FUNCTION AddToBundlesArray : BOOL
VAR_INPUT
	arr : POINTER TO Bundle;
	
END_VAR
VAR
END_VAR

FOR i:=0 TO CONSTS.maxQueue BY 1 DO
	IF BundleIsValid(bundlesQueue[i]) AND NOT bundlesBypass[i] THEN
		bundlesQueue[i] := bundleIn;
		bundlesBypass[i] := FALSE;
		
		receive := TRUE;
		RETURN;
	END_IF
END_FOR

END_FUNCTION

(* stored: Version 1.1.0.1, ProductVersion 3.1.4024.11
   POU AddToBundlesArray: Id {da469e5e-07e9-4d53-8efa-674a41b6607c}, SpecialFunc None *)
